(* IEC 61131-3 sources: repolevel_ST_code_completion/output/0121完整版本/repoeval_Decorator_Application/readful_result_before_fix, 8 files *)

(* ---- ConcreteComponment.st ---- *)
{attribute 'enable_dynamic_creation'}
//This class creates the most basic object well called. This object is to be decorated
FUNCTION_BLOCK ConcreteComponent IMPLEMENTS Component_Interface
VAR_INPUT
END_VAR
VAR_OUTPUT
END_VAR
VAR
	sDescription : STRING;
	rValue : REAL;
END_VAR

METHOD CreateObject : BOOL
VAR
	bSuccess : BOOL;
END_VAR

bSuccess := FALSE;

IF sDescription = '' THEN
	sDescription := 'Default Description';
END_IF;

IF rValue = 0.0 THEN
	rValue := 1.0;
END_IF;

bSuccess := TRUE;

CreateObject := bSuccess;
END_FUNCTION_BLOCK

(* ---- ConcreteDecoratorA.st ---- *)
{attribute 'enable_dynamic_creation'}
//This class acts as a decorating class. It adds responsibilities and functionality to the component
FUNCTION_BLOCK ConcreteDecoratorA EXTENDS Decorator
VAR_INPUT
	//Reference to store the component to be decorated
	tempInputComponent : Component_Interface;
END_VAR
VAR_OUTPUT
END_VAR
VAR
    //Local variables to store intermediate values
    sTempDescription : STRING;
    rTempValue : REAL;
END_VAR

tempComponent := tempInputComponent; //Assign the input component to the decorator's component reference

//Retrieve and modify the description
sTempDescription := tempComponent.GetDescription();
sDescription := CONCAT(sTempDescription, ' + DecoratorA');

//Retrieve and modify the value
rTempValue := tempComponent.GetValue();
rValue := rTempValue + 10.0; //Add specific functionality by increasing the value

RETURN;
END_FUNCTION_BLOCK

(* ---- ConcreteDecoratorB.st ---- *)
{attribute 'enable_dynamic_creation'}
//This class acts as a decorating class. It adds responsibilities and functionality to the component
FUNCTION_BLOCK ConcreteDecoratorB EXTENDS Decorator
VAR_INPUT
	//Reference to store the component to be decorated
	tempInputComponent : Component_Interface;
END_VAR
VAR_OUTPUT
END_VAR
VAR
    // Local variable to store the updated description
    sUpdatedDescription : STRING;
    // Local variable to store the updated value
    rUpdatedValue : REAL;
END_VAR

tempComponent := tempInputComponent;

// Update the description by appending additional functionality
sUpdatedDescription := tempComponent.GetDescription() + ' + DecoratorB Functionality';
sDescription := sUpdatedDescription;

// Update the value by adding additional functionality
rUpdatedValue := tempComponent.GetValue() + 10.0; // Example value addition
rValue := rUpdatedValue;
END_FUNCTION_BLOCK

(* ---- ConcreteDecoratorC.st ---- *)
{attribute 'enable_dynamic_creation'}
//This class acts as a decorating class. It adds responsibilities and functionality to the component
FUNCTION_BLOCK ConcreteDecoratorC EXTENDS Decorator
VAR_INPUT
	//Reference to store the component to be decorated
	tempInputComponent : Component_Interface;
END_VAR
VAR_OUTPUT
END_VAR
VAR
END_VAR

tempComponent := tempInputComponent;
sDescription := tempComponent.GetDescription() + ' with additional functionality from ConcreteDecoratorC';
rValue := tempComponent.GetValue() + 10.0;
END_FUNCTION_BLOCK

(* ---- ConcreteComponment_getDescription.st ---- *)
//Illustrative method of the pattern
METHOD getDescription : STRING
VAR_INPUT
END_VAR
VAR_OUTPUT
END_VAR
VAR
    // Variable to store the description of the object
    sDescription : STRING;
END_VAR

// Retrieve and return the description of the object
getDescription := sDescription;
END_OTHER

(* ---- ConcreteComponment_getValue.st ---- *)
//Illustrative method of the pattern
METHOD getValue : REAL
VAR_INPUT
END_VAR
VAR_OUTPUT
END_VAR
VAR
    rPlainValue : REAL;
END_VAR

rPlainValue := THIS^.rValue;
getValue := rPlainValue;
END_OTHER

(* ---- ConcreteDecoratorA_getDescription.st ---- *)
//Illustrative method of the pattern
METHOD getDescription : STRING
VAR_INPUT
	//Reference to store the component to be decorated
	tempInputComponent : Component_Interface;
END_VAR
VAR
	//Variable to save the state of the concrete component to be decorated
	tempComponent : Component_Interface;
	//String variable to save the Description of the component
	sDescription : STRING;
END_VAR

tempComponent := tempInputComponent;
sDescription := ' Decorator Description';
getDescription := CONCAT(tempComponent.getDescription(), sDescription);
END_OTHER

(* ---- ConcreteDecoratorA_getValue.st ---- *)
//Illustrative method of the pattern
METHOD getValue : REAL
VAR_INPUT
	//Reference to store the component to be decorated
	tempInputComponent : Component_Interface;
END_VAR
VAR_OUTPUT
END_VAR
VAR
	//Variable to save the state of the concrete component to be decorated
	tempComponent : Component_Interface;
	//Real variable to save the Value of the component
	rValue : REAL := 0.5; // Fixed decoration value
END_VAR

// Assign the input component to the temporary component variable
tempComponent := tempInputComponent;

// Outputs the decorated cost of the component by obtaining the cost of the component to be decorated
// stored in tempComponent.getValue() and then adds the decoration value (0.5 as example)
getValue := tempComponent.getValue() + rValue;
END_OTHER
